SUBAPPLICATION Ventilsteuerung_Uebung_009a (* RampLimitFS *)
  (* Standard: 61499-2 *)
  (* Version 1.0, 2023-10-23, franz *)
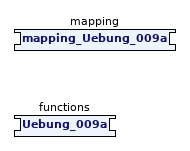
  SUBAPPS
    mapping : mapping_Uebung_009a;
    functions : Uebung_009a;
  END_SUBAPPS
END_SUBAPPLICATION
